// TIA Portal V19 export
VAR_GLOBAL   // PLC tag table "Standard-Variablentabelle"
   System_Byte AT %MB0 : Byte;
   FirstScan AT %M0.0 : Bool;
   DiagStatusUpdate AT %M0.1 : Bool;
   AlwaysTRUE AT %M0.2 : Bool;
   AlwaysFALSE AT %M0.3 : Bool;
   Clock_Byte AT %MB50 : Byte;
   Clock_10Hz AT %M50.0 : Bool;
   Clock_5Hz AT %M50.1 : Bool;
   "Clock_2.5Hz" AT %M50.2 : Bool;
   Clock_2Hz AT %M50.3 : Bool;
   "Clock_1.25Hz" AT %M50.4 : Bool;
   Clock_1Hz AT %M50.5 : Bool;
   "Clock_0.625Hz" AT %M50.6 : Bool;
   "Clock_0.5Hz" AT %M50.7 : Bool;
   MB_SystemAltTakt AT %MB51 : Byte;
   MB_Imp_ClockByte AT %MB52 : Byte;
   Imp_10Hz AT %M52.0 : Bool;
   Imp_5Hz AT %M52.1 : Bool;
   "Imp_2.5Hz" AT %M52.2 : Bool;
   Imp_2Hz AT %M52.3 : Bool;
   "Imp_1.25Hz" AT %M52.4 : Bool;
   Imp_1Hz AT %M52.5 : Bool;
   "Imp_0.625Hz" AT %M52.6 : Bool;
   "Imp_0.5Hz" AT %M52.7 : Bool;
   T_Verz_NotAus AT %T1 : Timer;
   T_ErrQuitt AT %T4 : Timer;   // Verlängerung Fehlerquittung für FUs
   T_Aend_WT AT %T5 : Timer;
   T_nAuto_TW_1 AT %T10 : Timer;   // Timer0 TW nicht in Automatik
   T_TO_Hub_TW_1_li AT %T11 : Timer;   // Timer1 TW Hub zu lange links
   T_TO_Fahrt_TW_1 AT %T12 : Timer;   // Timer2 TW Fahrt zu lange
   T_Laser_TW_1 AT %T13 : Timer;   // Timer3 TW Laser Request
   T_Speedout_TW_1 AT %T14 : Timer;   // Timer4 TW Speedout
   T_Verz_SU_TW_1 AT %T15 : Timer;   // Timer5 TW Verzögerung SU/SO
   T_Sim_SUL_TW_1 AT %T16 : Timer;   // Timer6 TW Simulation SUL
   T_TO_TS_TW_1 AT %T17 : Timer;   // Timer7 TW Tropfwanne zu lange
   T_TO_Hub_TW_1_re AT %T18 : Timer;   // Timer8 TW Hub zu lange rechts
   T_T9_TW_1 AT %T19 : Timer;   // Timer9 TW frei
   T_Verz_Auto AT %T210 : Timer;
   "T_Verzug StSpg" AT %T220 : Timer;   // Verzögerung Steuerspannung
   T_Hupe_Quitt_Auto AT %T255 : Timer;   // Timer für automatische Quittung der Hupe
   "T-TO-Komm-PNOZ" AT %T200 : Timer;
   T_Anlauf AT %T201 : Timer;
   temp_Sollzeit AT %MD256 : DInt;
   T_GO_links AT %T51 : Timer;
   T_GO_rechts AT %T52 : Timer;
   T_LS_vorn AT %T53 : Timer;
   T_LS_hinten AT %T54 : Timer;
   T_St_Last_links AT %T20 : Timer;
   T_St_Last_rechts AT %T21 : Timer;
   "TA-Pause_LF_CM01" AT %T31 : Timer;
   "TA-Pause_LF_CM02" AT %T32 : Timer;
   T_MobielPanel_Lebensbit_ein AT %T55 : Timer;
   T_MobielPanel_Lebensbit_aus AT %T56 : Timer;
   T_VEW_niO AT %T33 : Timer;
   GrossoptikIstAngefordert AT %M400.0 : Bool;
END_VAR
VAR_GLOBAL CONSTANT   // user constants
   WT_Typ_KS : Byte := B#16#11;   // kurz schmal
   WT_Typ_LS : Byte := B#16#12;   // lang schmal
   WT_Typ_GO : Byte := B#16#20;   // GroßOptik
   Anzahl_Alarm_Woerter : Int := 40;
   KorbAnzahl_min : Int := 1;
   KorbAnzahl_max : Int := 13;
END_VAR
